// TwinCAT 3 PLC project Untitled1
// ProgramVersion: 3.1.4024.0
// libraries:
//   Tc2_Standard, * (Beckhoff Automation GmbH)
//   Tc2_System, * (Beckhoff Automation GmbH)
//   Tc2_TcpIp, * (Beckhoff Automation GmbH)
//   Tc3_Module, * (Beckhoff Automation GmbH)
// project tree:
//   / PlcTask.TcTTO (not stored)
//   POUs/AmeClient/ AmeClient.TcPOU, AmeClientParam.TcGVL (not stored)
//   POUs/AmeClient/DUTs/AssyMethods/ St_Assy_Base.TcDUT, St_Assy_Complete.TcDUT, St_Assy_GetDetails.TcDUT (not stored), St_Assy_SetParametricsAndNCNative.TcDUT (not stored), St_Assy_SetReferences.TcDUT, St_Assy_SignOff.TcDUT (not stored), St_Assy_Start.TcDUT (not stored)
//   POUs/AmeClient/DUTs/ E_AssyComplete.TcDUT (not stored)
//   POUs/ MAIN.TcPOU (not stored)
//   POUs/OOP/ I_Command.TcIO, I_Device.TcIO (not stored), Stereo.TcPOU (not stored), TurnOffCommand.TcPOU, TurnOnCommand.TcPOU
// real-time tasks:
//   TASK PlcTask: cycle T#10ms, priority 20, ADS port 350

// ---- POUs/AmeClient/DUTs/AssyMethods/St_Assy_Base.TcDUT
TYPE St_Assy_Base :
STRUCT
	sSfc		:STRING;
	iOpIndex	:INT;
END_STRUCT
END_TYPE

// ---- POUs/AmeClient/DUTs/AssyMethods/St_Assy_Complete.TcDUT
TYPE St_Assy_Complete EXTENDS St_Assy_Base :
STRUCT
	eState		:E_AssyComplete;
END_STRUCT
END_TYPE

// ---- POUs/AmeClient/DUTs/AssyMethods/St_Assy_SetReferences.TcDUT
TYPE St_Assy_SetReferences EXTENDS St_Assy_Base :
STRUCT
	sCustomField	:STRING;
END_STRUCT
END_TYPE

// ---- POUs/OOP/I_Command.TcIO
INTERFACE I_Command

METHOD execute
END_METHOD

END_INTERFACE

// ---- POUs/AmeClient/AmeClient.TcPOU
FUNCTION_BLOCK AmeClient

VAR_OUTPUT
	bError	:BOOL;
END_VAR

VAR		// FB_Init
	_sType			:STRING(5) := '0';	
	_sSrvNetId		:T_AmsNetId;
	_sRemoteHost	:T_IPv4Addr;
	_udiRemotePort	:UDINT;
	_tTimeout		:TIME;
	_udiMsgSize		:UDINT;
END_VAR

VAR	
	_hSocket    		:T_HSOCKET;
	_sSendMsg			:STRING(AmeClientParam.udiMSG_SIZE);
	_sRcvMsg			:STRING(AmeClientParam.udiMSG_SIZE);
	_udiErrorSocketConn	:UDINT;
	_udiErrorSocketSend	:UDINT;
	_udiErrorSocketRcv	:UDINT;
	
	_bMethodInit		:BOOL;
	
	_sSeparator			:STRING(1) 	:= '|';
	
	_eStateM		:(
						IDLE := 0,
						EVALUATE_MSG,
						OPEN_CONNECTION,
						WAITING_FOR_CONNECTION,
						SEND_MSG,
						WAITTING_FOR_SEND_MSG,
						RCV_MSG,
						WAITTING_FOR_RCV_MSG,
						COPY_RCV_MSG,
						DONE,
						ERROR
						);
	_eError		:(
						NO_ERROR :=0,
						MSG_CANNOT_BE_EMPTY,
						CONNECTION_ERROR,
						SEND_MSG_ERROR,
						RCV_MSG_ERROR
						);
END_VAR

METHOD PUBLIC Assy_Complete_3011 :BOOL;
VAR_INPUT
	In	:St_Assy_Complete;
END_VAR

VAR
	_sActionCall	:STRING(4) 	:= '3011';
END_VAR
IF THIS^._bMethodInit = FALSE THEN
	THIS^.MethodInit();
	
	THIS^._sSendMsg := CONCAT(THIS^._sSendMsg, THIS^._sType);
	THIS^._sSendMsg := CONCAT(THIS^._sSendMsg, THIS^._sSeparator);
	This^._sSendMsg := CONCAT(This^._sSendMsg, _sActionCall);
	THIS^._sSendMsg := CONCAT(THIS^._sSendMsg, THIS^._sSeparator);
	THIS^._sSendMsg := CONCAT(THIS^._sSendMsg, In.sSfc);
	THIS^._sSendMsg := CONCAT(THIS^._sSendMsg, THIS^._sSeparator);
	THIS^._sSendMsg := CONCAT(THIS^._sSendMsg, INT_TO_STRING(In.eState));
	THIS^._sSendMsg := CONCAT(THIS^._sSendMsg, THIS^._sSeparator);
	THIS^._sSendMsg := CONCAT(THIS^._sSendMsg, INT_TO_STRING(In.iOpIndex));
	
	THIS^._bMethodInit := TRUE;
END_IF

IF THIS^._eError = NO_ERROR THEN
	IF THIS^._bMethodInit = TRUE AND_THEN  THIS^.SendRcvMsg()= TRUE THEN
		Assy_Complete_3011 		:= TRUE;
		THIS^._bMethodInit 	:= FALSE;
	END_IF
ELSE
	Assy_Complete_3011 		:= TRUE;
	THIS^._bMethodInit 	:= FALSE;
	THIS^.bError 		:= TRUE;
END_IF
END_METHOD

METHOD PUBLIC Assy_GetDetails_1026 :BOOL;
VAR_INPUT
	In	:St_Assy_GetDetails;
END_VAR

VAR
	_sActionCall	:STRING(4) 	:= '1026';
END_VAR
IF THIS^._bMethodInit = FALSE THEN
	THIS^.MethodInit();
	
	THIS^._sSendMsg := CONCAT(THIS^._sSendMsg, THIS^._sType);
	THIS^._sSendMsg := CONCAT(THIS^._sSendMsg, THIS^._sSeparator);
	THIS^._sSendMsg := CONCAT(THIS^._sSendMsg, _sActionCall);
	THIS^._sSendMsg := CONCAT(THIS^._sSendMsg, THIS^._sSeparator);
	THIS^._sSendMsg := CONCAT(THIS^._sSendMsg, In.sSfc);
	THIS^._sSendMsg := CONCAT(THIS^._sSendMsg, THIS^._sSeparator);
	THIS^._sSendMsg := CONCAT(THIS^._sSendMsg, INT_TO_STRING(In.iOpIndex));
	
	THIS^._bMethodInit := TRUE;
END_IF

IF THIS^._eError = NO_ERROR THEN
	IF THIS^._bMethodInit = TRUE AND_THEN  THIS^.SendRcvMsg()= TRUE THEN
		Assy_GetDetails_1026 := TRUE;
		THIS^._bMethodInit 	:= FALSE;
	END_IF
ELSE
	Assy_GetDetails_1026 	:= TRUE;
	THIS^._bMethodInit 	:= FALSE;
	THIS^.bError 		:= TRUE;
END_IF
END_METHOD

METHOD PUBLIC Assy_SetParametricsAndNCNative_3503 :BOOL;
VAR_INPUT
	In	:St_Assy_SetParametricsAndNCNative;
END_VAR
VAR
	_sActionCall		:STRING(4) 	:= '3503';	
END_VAR
IF THIS^._bMethodInit = FALSE THEN
	THIS^.MethodInit();
	
	THIS^._sSendMsg := CONCAT(THIS^._sSendMsg, THIS^._sType);
	THIS^._sSendMsg := CONCAT(THIS^._sSendMsg, THIS^._sSeparator);
	This^._sSendMsg := CONCAT(This^._sSendMsg, _sActionCall);
	THIS^._sSendMsg := CONCAT(THIS^._sSendMsg, THIS^._sSeparator);
	THIS^._sSendMsg := CONCAT(THIS^._sSendMsg, In.sSfc);
	THIS^._sSendMsg := CONCAT(THIS^._sSendMsg, THIS^._sSeparator);
	THIS^._sSendMsg := CONCAT(THIS^._sSendMsg, In.sProgramId);
	THIS^._sSendMsg := CONCAT(THIS^._sSendMsg, THIS^._sSeparator);
	THIS^._sSendMsg := CONCAT(THIS^._sSendMsg, In.sProgramRevision);
	THIS^._sSendMsg := CONCAT(THIS^._sSendMsg, THIS^._sSeparator);
	THIS^._sSendMsg := CONCAT(THIS^._sSendMsg, THIS^._sSeparator);
	THIS^._sSendMsg := CONCAT(THIS^._sSendMsg, THIS^._sSeparator);
	THIS^._sSendMsg := CONCAT(THIS^._sSendMsg, In.sTestStep);
	THIS^._sSendMsg := CONCAT(THIS^._sSendMsg, THIS^._sSeparator);
	THIS^._sSendMsg := CONCAT(THIS^._sSendMsg, THIS^._sSeparator);
	THIS^._sSendMsg := CONCAT(THIS^._sSendMsg, In.sDescription);
	THIS^._sSendMsg := CONCAT(THIS^._sSendMsg, THIS^._sSeparator);
	THIS^._sSendMsg := CONCAT(THIS^._sSendMsg, THIS^._sSeparator);
	THIS^._sSendMsg := CONCAT(THIS^._sSendMsg, In.sValue);
	THIS^._sSendMsg := CONCAT(THIS^._sSendMsg, THIS^._sSeparator);
	THIS^._sSendMsg := CONCAT(THIS^._sSendMsg, THIS^._sSeparator);
	THIS^._sSendMsg := CONCAT(THIS^._sSendMsg, In.sUnit);
	THIS^._sSendMsg := CONCAT(THIS^._sSendMsg, THIS^._sSeparator);
	THIS^._sSendMsg := CONCAT(THIS^._sSendMsg, THIS^._sSeparator);
	THIS^._sSendMsg := CONCAT(THIS^._sSendMsg, In.sLowerLimit);
	THIS^._sSendMsg := CONCAT(THIS^._sSendMsg, THIS^._sSeparator);
	THIS^._sSendMsg := CONCAT(THIS^._sSendMsg, THIS^._sSeparator);
	THIS^._sSendMsg := CONCAT(THIS^._sSendMsg, In.sUpperLimit);
	THIS^._sSendMsg := CONCAT(THIS^._sSendMsg, THIS^._sSeparator);
	THIS^._sSendMsg := CONCAT(THIS^._sSendMsg, THIS^._sSeparator);
	THIS^._sSendMsg := CONCAT(THIS^._sSendMsg, In.sState);
	THIS^._sSendMsg := CONCAT(THIS^._sSendMsg, THIS^._sSeparator);
	THIS^._sSendMsg := CONCAT(THIS^._sSendMsg, THIS^._sSeparator);
	THIS^._sSendMsg := CONCAT(THIS^._sSendMsg, In.sAdapter);
	THIS^._sSendMsg := CONCAT(THIS^._sSendMsg, THIS^._sSeparator);
	THIS^._sSendMsg := CONCAT(THIS^._sSendMsg, THIS^._sSeparator);
	THIS^._sSendMsg := CONCAT(THIS^._sSendMsg, THIS^._sSeparator);
	THIS^._sSendMsg := CONCAT(THIS^._sSendMsg, INT_TO_STRING(In.iOpIndex));
	
	THIS^._bMethodInit := TRUE;
END_IF

IF THIS^._eError = NO_ERROR THEN
	IF THIS^._bMethodInit = TRUE AND_THEN  THIS^.SendRcvMsg()= TRUE THEN
		Assy_SetParametricsAndNCNative_3503 	:= TRUE;
		THIS^._bMethodInit 				:= FALSE;
	END_IF
ELSE
	Assy_SetParametricsAndNCNative_3503 	:= TRUE;
	THIS^._bMethodInit 	:= FALSE;
	THIS^.bError 		:= TRUE;
END_IF
END_METHOD

METHOD PUBLIC Assy_SetReferences_3026 :BOOL;
VAR_INPUT
	In	:St_Assy_SetReferences;
END_VAR
VAR
	_sActionCall	:STRING(4) 	:= '3026';
END_VAR
IF THIS^._bMethodInit = FALSE THEN
	THIS^.MethodInit();	
	
	THIS^._sSendMsg := CONCAT(THIS^._sSendMsg, THIS^._sType);
	THIS^._sSendMsg := CONCAT(THIS^._sSendMsg, THIS^._sSeparator);
	THIS^._sSendMsg := CONCAT(THIS^._sSendMsg, _sActionCall);
	THIS^._sSendMsg := CONCAT(THIS^._sSendMsg, THIS^._sSeparator);
	THIS^._sSendMsg := CONCAT(THIS^._sSendMsg, In.sSfc);
	THIS^._sSendMsg := CONCAT(THIS^._sSendMsg, THIS^._sSeparator);
	THIS^._sSendMsg := CONCAT(THIS^._sSendMsg, In.sCustomField);
	THIS^._sSendMsg := CONCAT(THIS^._sSendMsg, THIS^._sSeparator);
	THIS^._sSendMsg := CONCAT(THIS^._sSendMsg, INT_TO_STRING(In.iOpIndex));
	
	THIS^._bMethodInit := TRUE;
END_IF

IF THIS^._eError = NO_ERROR THEN
	IF THIS^._bMethodInit = TRUE AND_THEN  THIS^.SendRcvMsg()= TRUE THEN
		Assy_SetReferences_3026 	:= TRUE;
		THIS^._bMethodInit 	:= FALSE;
	END_IF
ELSE
	Assy_SetReferences_3026 	:= TRUE;
	THIS^._bMethodInit 	:= FALSE;
	THIS^.bError 		:= TRUE;
END_IF
END_METHOD

METHOD PUBLIC Assy_SignOff :BOOL;
VAR_INPUT
	In	:St_Assy_SignOff;
END_VAR

VAR
	_sActionCall	:STRING(4) 	:= '3007';
END_VAR
IF THIS^._bMethodInit = FALSE THEN
	THIS^.MethodInit();
	
	THIS^._sSendMsg := CONCAT(THIS^._sSendMsg, THIS^._sType);
	THIS^._sSendMsg := CONCAT(THIS^._sSendMsg, THIS^._sSeparator);
	THIS^._sSendMsg := CONCAT(THIS^._sSendMsg, _sActionCall);
	THIS^._sSendMsg := CONCAT(THIS^._sSendMsg, THIS^._sSeparator);
	THIS^._sSendMsg := CONCAT(THIS^._sSendMsg, In.sSfc);
	THIS^._sSendMsg := CONCAT(THIS^._sSendMsg, THIS^._sSeparator);
	THIS^._sSendMsg := CONCAT(THIS^._sSendMsg, INT_TO_STRING(In.iOpIndex));
	
	THIS^._bMethodInit := TRUE;
END_IF

IF THIS^._eError = NO_ERROR THEN
	IF THIS^._bMethodInit = TRUE AND_THEN  THIS^.SendRcvMsg()= TRUE THEN
		Assy_SignOff 		:= TRUE;
		THIS^._bMethodInit 	:= FALSE;
	END_IF
ELSE
	Assy_SignOff 		:= TRUE;
	THIS^._bMethodInit 	:= FALSE;
	THIS^.bError 		:= TRUE;
END_IF
END_METHOD

METHOD PUBLIC Assy_Start :BOOL;
VAR_INPUT
	In	:St_Assy_Start;
END_VAR

VAR
	_sActionCall	:STRING(4) 	:= '3010';
END_VAR
IF THIS^._bMethodInit = FALSE THEN
	THIS^.MethodInit();
	
	THIS^._sSendMsg := CONCAT(THIS^._sSendMsg, THIS^._sType);
	THIS^._sSendMsg := CONCAT(THIS^._sSendMsg, THIS^._sSeparator);
	This^._sSendMsg := CONCAT(This^._sSendMsg, _sActionCall);
	THIS^._sSendMsg := CONCAT(THIS^._sSendMsg, THIS^._sSeparator);
	THIS^._sSendMsg := CONCAT(THIS^._sSendMsg, In.sSfc);
	THIS^._sSendMsg := CONCAT(THIS^._sSendMsg, THIS^._sSeparator);
	THIS^._sSendMsg := CONCAT(THIS^._sSendMsg, INT_TO_STRING(In.iOpIndex));
	
	_bMethodInit := TRUE;
END_IF

IF THIS^._eError = NO_ERROR THEN
	IF THIS^._bMethodInit = TRUE AND_THEN  THIS^.SendRcvMsg()= TRUE THEN
		Assy_Start 			:= TRUE;
		THIS^._bMethodInit 	:= FALSE;
	END_IF
ELSE
	Assy_Start 			:= TRUE;
	THIS^._bMethodInit 	:= FALSE;
	THIS^.bError 		:= TRUE;
END_IF
END_METHOD

METHOD FB_init : BOOL
VAR_INST
	//_SocketClose	:FB_SocketClose;
END_VAR
VAR_INPUT
	bInitRetains 	: BOOL; // if TRUE, the retain variables are initialized (warm start / cold start)
	bInCopyCode 	: BOOL;  // if TRUE, the instance afterwards gets moved into the copy code (online change)
	
	iType			:INT;
	sSrvNetId		:T_AmsNetId;
	sRemoteHost		:T_IPv4Addr;
	udiRemotePort	:UDINT;
	tTimeout		:TIME;
END_VAR
THIS^._sType 		:= INT_TO_STRING(iType);
THIS^._sSrvNetId	:= sSrvNetId;
THIS^._sRemoteHost	:= sRemoteHost;
THIS^._udiRemotePort:= udiRemotePort;

IF tTimeout <= T#0S THEN
	THIS^._tTimeout	:= DEFAULT_ADS_TIMEOUT;
ELSE
	THIS^._tTimeout	:= tTimeout;
END_IF
END_METHOD

METHOD PROTECTED MethodInit
VAR_INPUT
END_VAR
bError 		:= FALSE;
_eStateM 	:= IDLE;
_eError		:= NO_ERROR;
_sSendMsg 	:= '';
END_METHOD

METHOD PROTECTED SendRcvMsg :BOOL;
VAR_INPUT
END_VAR

VAR_INST
	_SocketConnect 		:FB_SocketConnect;
	_SocketSend			:FB_SocketSend;
	_SocketReceive		:FB_SocketReceive;
	_bOpenConn			:BOOL;
	_bSendMsg			:BOOL;
	_bRcvMsg			:BOOL;
	_iRecBytes			:INT;
	
END_VAR

VAR CONSTANT
	//_udiMAX_RCV_LENGHT	:UDINT :=4294967295;
END_VAR
//DESCRIPTION ************************************************
//************************************************************

CASE _eStateM OF
	IDLE:
		_eStateM := EVALUATE_MSG;
		
	EVALUATE_MSG:
		IF(_sSendMsg = '')
		THEN
			_eError 		:= MSG_CANNOT_BE_EMPTY;
			_eStateM := ERROR;
			
		ELSIF(_sSendMsg <> '')
		THEN
			_eError 		:= NO_ERROR;
			_eStateM	:= OPEN_CONNECTION;
		END_IF
		
	OPEN_CONNECTION:
		_bOpenConn	:= TRUE;
		
		IF (_SocketConnect.bError = TRUE)THEN
			_udiErrorSocketConn	:= _SocketConnect.nErrId;
			_eError				:= CONNECTION_ERROR;
			_eStateM 			:= ERROR;
			
		ELSIF(_SocketConnect.bBusy = TRUE AND _SocketConnect.bError = FALSE) THEN
			_eStateM := WAITING_FOR_CONNECTION;
		END_IF
		
	WAITING_FOR_CONNECTION:
		IF(_SocketConnect.bError = TRUE) THEN
			_udiErrorSocketConn	:= _SocketConnect.nErrId;
			_eError				:= CONNECTION_ERROR;
			_eStateM 			:= ERROR;
			
		ELSIF(_SocketConnect.bBusy = FALSE AND _SocketConnect.bError = FALSE) THEN
			_eStateM := SEND_MSG;
		END_IF
		
	SEND_MSG:
		_bSendMsg := TRUE;
		
		IF(_SocketSend.bBusy = TRUE)
		THEN
			_eStateM := WAITTING_FOR_SEND_MSG;
		END_IF
		
	WAITTING_FOR_SEND_MSG:
		IF(_SocketSend.bError = TRUE)
		THEN
			_udiErrorSocketSend 	:= _SocketSend.nErrId;
			_eError				:= SEND_MSG_ERROR;
			_eStateM 		:= ERROR;
		ELSIF(_SocketSend.bBusy = FALSE AND _SocketSend.bError = FALSE)
		THEN
			_eStateM := RCV_MSG;
		END_IF
		
	RCV_MSG:
		_bRcvMsg := TRUE;
		
		IF(_SocketReceive.bBusy = TRUE)
		THEN
			_eStateM := WAITTING_FOR_RCV_MSG;
		END_IF
		
	WAITTING_FOR_RCV_MSG:
		IF(_SocketReceive.bError = TRUE)
		THEN
			_udiErrorSocketRcv 	:= _SocketReceive.nErrId;
			_eError				:= RCV_MSG_ERROR;
			_eStateM 		:= ERROR;
			
		ELSIF(_SocketReceive.bBusy = FALSE AND _SocketReceive.bError = FALSE)
		THEN
			_eStateM := COPY_RCV_MSG;
		END_IF
	
	COPY_RCV_MSG:
		_iRecBytes		:= UDINT_TO_INT(_SocketReceive.nRecBytes);
		_sRcvMsg 		:= LEFT(_sRcvMsg,_iRecBytes);
		_eStateM 	:= DONE;
		
	DONE:
		_bOpenConn	:= FALSE;
		_bSendMsg	:= FALSE;
		_bRcvMsg	:= FALSE;
		
		SendRcvMsg	:= TRUE;
			
	ERROR:
		_bOpenConn	:= FALSE;
		_bSendMsg	:= FALSE;
		_bRcvMsg	:= FALSE;
		
		SendRcvMsg	:= TRUE;
		 	
END_CASE

_SocketConnect(
				sSrvNetId	:= _sSrvNetId, 
				sRemoteHost	:= _sRemoteHost, 
				nRemotePort	:= _udiRemotePort, 
				bExecute	:= _bOpenConn, 
				tTimeout	:= _tTimeout,  
				hSocket		=> _hSocket);
				            
_SocketSend(                 
				sSrvNetId	:= _sSrvNetId, 
				hSocket		:= _hSocket, 
				cbLen		:= INT_TO_UDINT(LEN(_sSendMsg)), 
				pSrc		:= ADR(_sSendMsg), 
				bExecute	:= _bSendMsg, 
				tTimeout	:= _tTimeout);
				            
_SocketReceive(              
				sSrvNetId	:= _sSrvNetId, 
				hSocket		:= _hSocket, 
				cbLen		:= AmeClientParam.udiMSG_SIZE, 
				pDest		:= ADR(_sRcvMsg), 
				bExecute	:= _bRcvMsg, 
				tTimeout	:= _tTimeout);
END_METHOD

PROPERTY PUBLIC sRcvMsg : STRING
GET
sRcvMsg	:= _sRcvMsg;
END_GET
END_PROPERTY

PROPERTY PUBLIC sSendMsg : STRING
GET
sSendMsg := _sSendMsg;
END_GET
END_PROPERTY

END_FUNCTION_BLOCK

// ---- POUs/OOP/TurnOffCommand.TcPOU
FUNCTION_BLOCK TurnOffCommand EXTENDS I_Command
VAR
	_device	:I_Device;
END_VAR

METHOD execute
_device.turnOff();
END_METHOD

METHOD FB_init : BOOL
VAR_INPUT
	bInitRetains : BOOL; // if TRUE, the retain variables are initialized (warm start / cold start)
	bInCopyCode : BOOL;  // if TRUE, the instance afterwards gets moved into the copy code (online change)
	
	device	:I_Device;
END_VAR
THIS^._device := device;
END_METHOD

END_FUNCTION_BLOCK

// ---- POUs/OOP/TurnOnCommand.TcPOU
FUNCTION_BLOCK TurnOnCommand EXTENDS I_Command
VAR
	_device	:I_Device;
END_VAR

METHOD execute
_device.turnOn();
END_METHOD

METHOD FB_init : BOOL
VAR_INPUT
	bInitRetains : BOOL; // if TRUE, the retain variables are initialized (warm start / cold start)
	bInCopyCode : BOOL;  // if TRUE, the instance afterwards gets moved into the copy code (online change)
	
	device	:I_Device;
END_VAR
This^._device := device;
END_METHOD

END_FUNCTION_BLOCK
